# B&R Automation Studio project Lab3
Automation Studio 4.5.2.102

## Configuration Config1

### Task classes (Cpu.sw)
```
Cyclic#4:
  Program <- Program.prg
Libraries: Acp10man, Acp10par, NcGlobal, Library
```

### IoMap.iom - 4PP065_0571_P74/IoMap.iom
```iecst
VAR_CONFIG
	Cyclic#1.gAxis01_DrvIf.iDrvOK AT %IX."8I64xxxxxxx.00x-1".ETAD_Input_Bool_02;
	Cyclic#1.::Program:speed AT %QW."8I64xxxxxxx.00x-1".LFRD_Output;
	Cyclic#1.gAxis01_DiDoIf.oDriveEnable AT %QX."8I64xxxxxxx.00x-1".CMDD_Output_Bool_00;
	Cyclic#1.gAxis01_ModuleOk AT %QX."8I64xxxxxxx.00x-1".CMDD_Output_Bool_01;
	Cyclic#1.gAxis01_ModuleOk AT %QX."8I64xxxxxxx.00x-1".CMDD_Output_Bool_02;
	Cyclic#1.gAxis01_DiDoIf.oDriveEnable AT %QX."8I64xxxxxxx.00x-1".CMDD_Output_Bool_03;
	Cyclic#1.gAxis01_DiDoIf.iDriveReady AT %IX."8I64xxxxxxx.00x-1".ETAD_Input_Bool_02;
	::Program:EVIRD.STATE AT %IW."8I64xxxxxxx.00x-1".ETAD_Input;
	::Program:EVIRD.COM AT %QW."8I64xxxxxxx.00x-1".CMDD_Output;
END_VAR
```

### Acp10map.ncm - 4PP065_0571_P74/Motion/Acp10map.ncm
```
NcMapping (NcSwId=Acp10)
  NcObject gAxis01 (ModuleId=8I64xxxxxxx.00x-1, ModuleAddress=SDC_IF1.ST3, Type=ncAXIS, Channel=1, AcoposSimulation=Off, InitParameter=gAxis01i, AcoposParameter=gAxis01a, Disabled=FALSE, ModuleDisabled=FALSE)
```

## Logical view

### Library Logical/Libraries/Library

#### Library.fun
```iecst
{REDUND_ERROR} FUNCTION_BLOCK DRIVE (*TODO: Add your comment here*) (*$GROUP=User,$CAT=User,$GROUPICON=User.png,$CATICON=User.png*)
	VAR_INPUT
		STATE : UINT;
		enable : BOOL;
	END_VAR
	VAR_OUTPUT
		COM : UINT;
	END_VAR
END_FUNCTION_BLOCK
```

#### DRIVE.c
```c
#include <bur/plctypes.h>
#ifdef __cplusplus
	extern "C"
	{
#endif
	#include "Library.h"
#ifdef __cplusplus
	};
#endif
/* TODO: Add your comment here */
void DRIVE(struct DRIVE* inst)
{
	UINT mask=inst->STATE & 0x6f;
	if (!inst->enable)
	{
		inst->COM = CMD_SHUTDOWN;
	}
	else
	{
		switch(mask)
		{
			case STATE_DISABLED:
				inst->COM=CMD_SHUTDOWN;
				break;

			case STATE_READY:
				inst->COM=CMD_ENABLED;
				break;

			case STATE_SWITCHED_ON:
				inst->COM=CMD_SWITCHED_ON;
				break;
		}
	}
}
```

### Program Logical/Program

#### Variables.var
```iecst
VAR
	speed : INT;
	EVIRD : DRIVE;
END_VAR
```

#### Main.c
```c
#include <bur/plctypes.h>

#ifdef _DEFAULT_INCLUDES
	#include <AsDefault.h>
#endif

void _INIT ProgramInit(void)
{
	speed = 100;
	EVIRD.enable=1;
}

void _CYCLIC ProgramCyclic(void)
{
	DRIVE(&EVIRD);
}

void _EXIT ProgramExit(void)
{

}
```
